FUNCTION F_TargetWindowReachedAxisRef : BOOL
VAR_IN_OUT
	/// Achse als Referenz
	fbAxis		:FB_AxisDriver;
END_VAR
VAR_INPUT
	fTargetPos: LREAL;
	fWindow: LREAL;
END_VAR


F_TargetWindowReachedAxisRef := fbAxis.Position >= (fTargetPos - fWindow) AND fbAxis.Position <= (fTargetPos + fWindow);

END_FUNCTION

(* stored: Version 1.1.0.1, ProductVersion 3.1.4020.12
   POU F_TargetWindowReachedAxisRef: Id {61062702-2c06-46f5-a7ac-a9c37e4bd3ab}, SpecialFunc None *)
